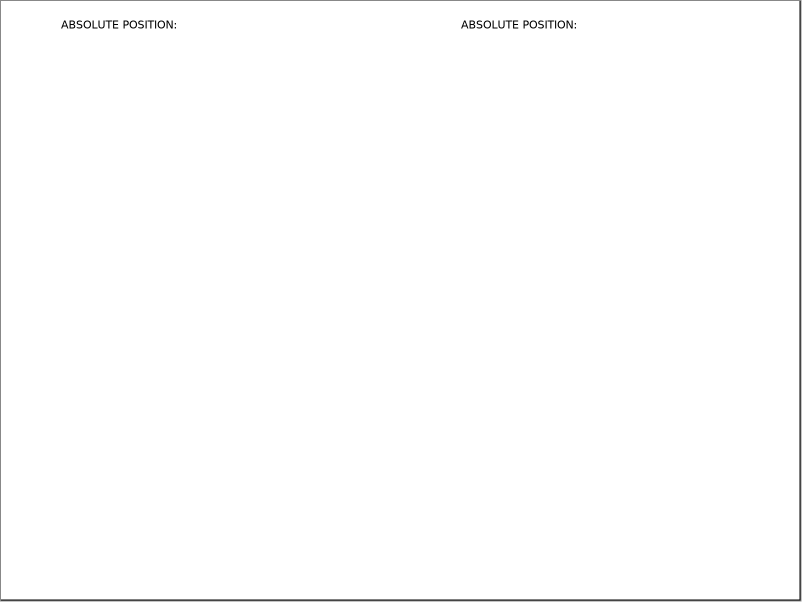
VISUALIZATION F49_Cam_Scaling  // 802x602
    Rectangle (0,0 800x600)
    Label (10,10 170x30), "ABSOLUTE POSITION:"
    Label (410,10 170x30), "ABSOLUTE POSITION:"
END_VISUALIZATION

(* stored: Version 1.1.0.1, ProductVersion 3.1.4022.7
   Visu F49_Cam_Scaling: Id {68c490c0-f404-439f-a433-83b12e13e96f} *)
